Universal Robots PolyScope program: TEST_SUB_121.urp

Program TEST_SUB_121 (installation=GD directory=/programs/GD createdIn=5.13.0 lastSavedIn=5.13.0 robotSerialNumber=20205000017)
Calibrated DH parameters: a=[-0.000157, -0.56303, -0.236706, -0.000074, -0.000109, 0]; d=[0.181705, 47.632387, 369.599619, -417.058513, 0.119878, 0.115667]; alpha=[1.570881, -0.005074, -0.001247, 1.56886, -1.570997, 0]; deltaTheta=[0, -0.405485, 5.544791, 1.143886, -0.000009, -0.000001]
InitVariablesNode
BeforeStart
  Script file /programs/GD/CONTROL/ALIGN_AXIS.script
    | def GET_NORM_VEC(p,axis=2):
    |   rot=p[0.0, 0.0, 0.0, p[3], p[4], p[5]]
    |   vec=p[0.0, 0.0, 0.0, 0.0, 0.0, 0.0]
    |   vec[axis]=1.0
    |   norm_p=pose_trans(rot,vec)
    |   return [norm_p[0], norm_p[1], norm_p[2]]
    | end
    | 
    | def GET_INNER_PRODUCT(v1,v2):
    |   return v1[0]*v2[0]+v1[1]*v2[1]+v1[2]*v2[2]
    | end
    | def GET_OUTER_PRODUCT(v1,v2):
    |   x=v1[1]*v2[2]-v1[2]*v2[1]
    |   y=v1[2]*v2[0]-v1[0]*v2[2]
    |   z=v1[0]*v2[1]-v1[1]*v2[0]
    |   return [x,y,z]
    | end
    | def GET_THETA(v1,v2):
    | #  cos=GET_INNER_PRODUCT(v1,v2) / norm(v1) / norm(v2)
    |   cos=GET_INNER_PRODUCT(v1,v2)
    |   g_cos=cos
    |   theta=norm(acos(cos))
    |   return theta
    | end
    | 
    | def GET_ALIGNED_POSE(target,feature,axis=2):
    |   feature_from_target=pose_trans(pose_inv(target),feature)
    |   g_f_from_t=feature_from_target
    |   nz_feature_from_target=GET_NORM_VEC(feature_from_target,axis)
    |   g_nz_f_from_t=nz_feature_from_target
    |   nz_target_from_target=[0.0, 0.0, 0.0]
    |   nz_target_from_target[axis]=1.0
    |   g_nz_t_from_t=nz_target_from_target
    | 
    |   theta=GET_THETA(nz_feature_from_target,nz_target_from_target)
    |   g_theta=theta
    |   rot_vec_n=normalize(GET_OUTER_PRODUCT(nz_target_from_target,nz_feature_from_target))
    | 
    |   if theta>d2r(90.0):
    |     theta=theta-d2r(180.0)
    |   end
    |   rot_vec=rot_vec_n * (theta)
    |   rot_p=p[0.0,0.0,0.0,rot_vec[0],rot_vec[1],rot_vec[2]]
    |   return pose_trans(target,rot_p)
    | end
    | def GET_ALIGNED_TCP(feature,axis=2):
    |   tcp=get_actual_tcp_pose()
    |   return GET_ALIGNED_POSE(tcp,feature,axis)
    | end
  Script file /programs/GD/CONTROL/ROTATE_CONTROL.script
    | def GET_TCP_FORCE_TOOL():
    |   force_torque=get_tcp_force()
    |   force_B=p[force_torque[0], force_torque[1], force_torque[2], 0, 0, 0]
    |   torque_B=p[force_torque[3], force_torque[4], force_torque[5], 0, 0, 0]
    |   tcp=get_actual_tcp_pose()
    |   rotation_BT=p[0, 0, 0, tcp[3], tcp[4], tcp[5]]
    |   force_T=pose_trans(pose_inv(rotation_BT), force_B)
    |   torque_T=pose_trans(pose_inv(rotation_BT), torque_B)
    |   force_torque_T=p[force_T[0], force_T[1], force_T[2], torque_T[0], torque_T[1], torque_T[2]]
    |   return force_torque_T
    | end
    | 
    | def GET_FORCE_VALUE_RZ(target):
    |   PoseSub= pose_sub (CurrPos_p,target)
    |   RZSub=r2d(PoseSub[5])
    |   if (RZSub<0):
    |     RZMin=-RZSupDegMin[0]
    |     RZRatio=RZSupRatio[0]
    |     RZOffset=-RZSupOffset[0]
    |   else:
    |     RZMin=-RZSupDegMin[1]
    |     RZRatio=RZSupRatio[1]
    |     RZOffset=RZSupOffset[1]
    |   end
    |   if (norm(RZSub) >= norm(RZMin)):
    |     RZSupForceVal=(RZMin-RZSub)*RZRatio+RZOffset
    |   else:
    |     RZSupForceVal=0
    |   end
    |   return RZSupForceVal
    | end
    | 
    | def GET_CVCORR_RZ(target):
    |   PoseSub=pose_sub(CurrPos_p,target)
    |   RYSub=r2d(PoseSub[4])
    |   if (RYSub<0):
    |     RYMin=-CVCorrDegMin[0]
    |     RZRatio=CVCorrRatio[0]
    |     RZOffset=-CVCorrOffset[0]
    |   else:
    |     RYMin=-CVCorrDegMin[1]
    |     RZRatio=CVCorrRatio[1]
    |     RZOffset=CVCorrOffset[1]
    |   end
    |   if (norm(RYSub) >= norm(RYMin)):
    |     CVCorrRZVal=RYSub*RZRatio+RZOffset
    |   else:
    |     CVCorrRZVal=0
    |   end
    |   return CVCorrRZVal
    | end
Robot Program (runOnlyOnce=true)
  Set NoAction tcp=TCP_1
  Script: sync()
  Script: CurrPos_p=get_actual_tcp_pose()
  CurrposAligned := p[0,0,0,0,0,0]
  CurrposAligned := GET_ALIGNED_TCP(CurrposAligned)
  RZSub := GET_CVCORR_RZ(CurrposAligned)
  Popup Message (haltProgram=false message=start! inputType=Text)
  MoveL speed 60 mm/s, acceleration 10 mm/s^2 (useActiveTCP=false) tcp=TCP_1; feature=Base
    If (norm(RZSub)≠0.0)
      PoseAdd := pose_add(p[0,0,0,0,0,d2r(-RZSub)],p[0,0,0,CurrPos_p[3],CurrPos_p[4],CurrPos_p[5]])
      PoseAdd := p[CurrPos_p[0],CurrPos_p[1],CurrPos_p[2],PoseAdd[3],PoseAdd[4],PoseAdd[5]]
      Waypoint Variable (Variable): variable=PoseAdd
  Popup Message (haltProgram=false message=done! inputType=Text)
Thread スレッド_1 (runOnlyOnce=false)
  Script: CurrPos_p=get_actual_tcp_pose()
